Universal Robots PolyScope program: RC_E8_PICK_820.urp

Program RC_E8_PICK_820 (createdIn=3.0.0 lastSavedIn=3.0.0 directory=/programs installation=default)
Robot Program (runOnlyOnce=true motionType=MoveJ speed=1.047198 acceleration=1.396263 useActiveTCP=false)
  'Program generated by RoboDK v4.1.0 for UR3e_HORNO on 05/09/2022 13:25:11'
  'Using nominal kinematics.'
  'Using Ref. Frame Traslado C: p[0.369000, -0.220000, 0.032000, 0.000000, 0.000000, 0.000000]'
  'Using TCP 0208-0001-0001-307-000-3 Horno: p[0.000000, 0.000000, 0.164750, 0.000000, 0.000000, 0.000000]'
  Script: set_tcp(p[0.000000, 0.000000, 0.164750, 0.000000, 0.000000, 0.000000])
  Script: movej([-0.418006, -2.151118, -0.151320, -2.416408, 1.600991, 4.345870],0.60000,0.12500,0,0.0000)
  Script: movej([-0.395125, -1.810392, -1.210131, -1.698044, 1.566184, 4.368573],0.05000,0.05000,0,0.0000)
  'Attach to 0208-0001-0001-307-000-3 Horno'
  MoveL speed 100 mm/s, acceleration 100 mm/s^2 (useActiveTCP=true)
    Waypoint Waypoint_1: TCP in base x=647.647 y=-478.682 z=288.936 mm, rx=-3.1102 ry=0.0802 rz=-0.0087 rad; joints [-23.95, -123.25, -8.67, -138.45, 91.73, 249] deg; flange x=646.6 y=-483.659 z=453.608 mm, rx=-3.1102 ry=0.0802 rz=-0.0087 rad
